Staubli VAL3: Wizard_smlBox.pgx

program Wizard_smlBox(string x_sName, num& x_nResult)
begin
  if set:bWizard
    call markTraj(x_nResult)
  endIf
  if x_nResult==0
    if set:bWizard
      call set:loadMarkData(x_sName,sMarkList)
    endIf
    if x_nResult==0
      call set:editSmlData(x_sName,x_nResult)
      if x_nResult==0
        call set:onSave()
      endIf
    endIf
  endIf

end
